TYPE E_PIZZA_TYPES :
(
	eType_Cheese := 0,
	eType_Pepperoni := 1,
	eType_Sausage := 2
);
END_TYPE

(* stored: Version 1.1.0.1, ProductVersion 3.1.0.26
   DUT E_PIZZA_TYPES: Id {c60bb2ba-c5ae-4915-8644-ae9b01f0c28d} *)
